// TIA Portal V17 export
// export: Created 2026-04-13T11:12:41.3915704Z, ExportSetting WithDefaults, DisplayName Totally Integrated Automation Portal, DisplayVersion V17 Update 4, DisplayName TIA Portal Openness, DisplayVersion V17 Update 4, DisplayName TIA Portal Version Control Interface, DisplayVersion V17, DisplayName SINAMICS Startdrive Advanced, DisplayVersion V17, DisplayName SINAMICS Startdrive G130, G150, S120, S150, SINAMICS MV, S210, DisplayVersion V17, DisplayName SINAMICS Startdrive G110M, G120, G120C, G120D, G120P, G115D, DisplayVersion V17, DisplayName STEP 7 Professional, DisplayVersion V17 Update 4, DisplayName STEP 7 Safety, DisplayVersion V17, DisplayName WinCC Professional, DisplayVersion V17 Update 4
FUNCTION_BLOCK "A1-台达DTC"   // FB33, SCL
{ S7_Optimized_Access := 'TRUE' }
VERSION : 0.1
// stored: AutoNumber true, IsIECCheckEnabled false, IsRetainMemResEnabled false, MemoryReserve 100, SetENOAutomatically false, UDAEnableTagReadback false
   VAR_INPUT
      站号 : UInt;
      触发 : Bool;
      输入模式 : Int;
      输入开关 : Bool;
      A输入设定 : Real;
      输入开度 : Real;
   END_VAR
   VAR_OUTPUT
      结束 : Bool;
      高高报警 : Bool;
      高报警 : Bool;
      低报警 : Bool;
      低低报警 : Bool;
      传感器故障 : Bool;
      输出控制P : Real;
      输出控制I : Real;
      输出控制D : Real;
      输出开度读 : Real;
   END_VAR
   VAR_IN_OUT
      B当前量 : Real;
      输入设定读 : Real;
      输出模式读 : Real;
      高高报设置 : Real;
      高报设置 : Real;
      低报设置 : Real;
      低低报设置 : Real;
      自整定开关 : Bool;
      Modbus_Master_Instance : Modbus_Master;
   END_VAR
   VAR DB_SPECIFIC
      当前指令ID : Int;
      上一次指令ID : Int;
      modbus_data : Struct
         触发 : Bool;
         站号 : UInt;
         模式 : USInt;
         地址 : UDInt;
         数据长度 : UInt;
         完成 : Bool;
         忙碌 : Bool;
         出错 : Bool;
         故障码 : Word;
         数据缓存区 : Array[1..50] of Word;
      END_STRUCT;
      报错代码 : Array[1..20] of Word;
      进温P读 : Int;
      进温I读 : Int;
      进温D读 : Int;
      T1_SV_写 : Int;
      进温AT开关 : Bool;
      进温AT开关_bak : Bool;
      进温AT_写字 : UInt;
      进温AT_读字 : UInt;
      T1_P值比对1 : Int;
      T1_P值比对2 : Int;
      进温启停字 : UInt;
      T1 { S7_SetPoint := 'True'} : TON_TIME;
   END_VAR
   VAR_TEMP
      tm_int : Int;
      tm_real : Real;
   END_VAR
BEGIN
   //程序1

   IF #触发 THEN
       #当前指令ID := 1;
   END_IF;

   #modbus_data.站号 := #站号;

   IF #当前指令ID = 9 THEN
       IF #进温AT_写字 = #进温AT_读字 THEN
           #当前指令ID := 10;
       END_IF;
   END_IF;

   CASE #当前指令ID OF
       1:
           //读取地址44097-44098
           #modbus_data.模式 := 0;
           #modbus_data.地址 := 44097;
           #modbus_data.数据长度 := 2;
       2:
           //读取地址44102
           (* 1005H-4101-44102  默认0   控制方式 0：PID；1：ON/OFF；2：手动；3：PID 过程控制 *)
           #modbus_data.模式 := 0;
           #modbus_data.地址 := 44102;
           #modbus_data.数据长度 := 1;
       3:
           //读取地址44106-44108
           (*  
           1009H-4105-44106  默认476 PB 比例带设定值 1 ~ 9,999, 温度单位为 0.1 度，模拟输入为 1EU
           100AH-4106-44107  默认260 Ti 积分控制常量设定值 0 ~ 9,999
           100BH-4107-44108  默认41 Td 微分控制常量设定值 0 ~ 9,999 *)
           #modbus_data.模式 := 0;
           #modbus_data.地址 := 44106;
           #modbus_data.数据长度 := 3;
       4:
           //读取地址44116
           (* 1013H-4115-44116  默认0   输出 2 输出量读取与写入 单位为 0.1%，写入只在手动控制模式下有效（DTC1000/2000 机种） *)
           #modbus_data.模式 := 0;
           #modbus_data.地址 := 44116;
           #modbus_data.数据长度 := 1;
       5:
           //读取地址12068
           (* 0813H-2067-12068  读写自动调谐状态 自动调谐停止：0（预设），自动调谐开始：1 *)
           #modbus_data.模式 := 0;
           #modbus_data.地址 := 12068;
           #modbus_data.数据长度 := 1;
       6:
           //写入地址44098
           (* 1001H-4097-44098       默认0 "SV" 设定值 温度以 0.1 度为计量单位，模拟输入为 1EU。 *)
           #tm_real := #A输入设定 * 10.0;
           #T1_SV_写 := REAL_TO_INT(#tm_real);
           #modbus_data.数据缓存区[1] := INT_TO_WORD(#T1_SV_写);
           #modbus_data.模式 := 1;
           #modbus_data.地址 := 44098;
           #modbus_data.数据长度 := 1;
       7:
           //写入地址44102
           (* 1005H-4101-44102  默认0   控制方式 0：PID；1：ON/OFF；2：手动；3：PID 过程控制 *)
           #modbus_data.数据缓存区[1] := INT_TO_WORD(#输入模式);
           #modbus_data.模式 := 1;
           #modbus_data.地址 := 44102;
           #modbus_data.数据长度 := 1;
       8:
           //写入地址44116
           (* 1013H-4115-44116  默认0   输出 2 输出量读取与写入 单位为 0.1%，写入只在手动控制模式下有效（DTC1000/2000 机种） *)
           #tm_real := #输入开度 * 10;
           #tm_int := REAL_TO_INT(#tm_real);
           #modbus_data.数据缓存区[1] := INT_TO_WORD(#tm_int);
           #modbus_data.模式 := 1;
           #modbus_data.地址 := 44116;
           #modbus_data.数据长度 := 1;
       9:
           //写入地址2068
           (* 0813H-2067-12068  读写自动调谐状态 自动调谐停止：0（预设），自动调谐开始：1 *)

           #modbus_data.数据缓存区[1] := UINT_TO_WORD(#进温AT_写字);
           #modbus_data.模式 := 1;
           #modbus_data.地址 := 2068;
           #modbus_data.数据长度 := 1;
       10:
           //写入地址2069
           (* 0814H-2068-12069  控制执行/停止设定 0：停止，1：执行（预设） *)
           #modbus_data.数据缓存区[1] := UINT_TO_WORD(#进温启停字);
           #modbus_data.模式 := 1;
           #modbus_data.地址 := 2069;
           #modbus_data.数据长度 := 1;

   END_CASE;




   #modbus_data.触发 := #当前指令ID <> #上一次指令ID;
   #上一次指令ID := #当前指令ID;



   //程序2


   #Modbus_Master_Instance(REQ := #modbus_data.触发,
                           MB_ADDR := #modbus_data.站号,
                           MODE := #modbus_data.模式,
                           DATA_ADDR := #modbus_data.地址,
                           DATA_LEN := #modbus_data.数据长度,
                           DONE => #modbus_data.完成,
                           BUSY => #modbus_data.忙碌,
                           ERROR => #modbus_data.出错,
                           STATUS => #modbus_data.故障码,
                           DATA_PTR := #modbus_data.数据缓存区);

   //程序3

   IF #modbus_data.完成 THEN
       CASE #当前指令ID OF
           1:
               //44097
               (* 1000H-4096-44097       PV 目前测量值
               （温度以 0.1 刻度为计量单位，模拟输入为 1EU。
               下列读值表示错误发生：
               8002H（32770） 输入读值尚未取得
               8003H（32771） 未接传感器
               8004H（32772） 传感器型式错误
               8006H（34774） 输入值无法测量,输入 ADC 错误
               8007H（32775） 内存无法读写） *)
               #tm_int := WORD_TO_INT(#modbus_data.数据缓存区[1]);
               #tm_real := INT_TO_REAL(#tm_int);
               #B当前量 := #tm_real / 10;
               //44098
               #tm_int := WORD_TO_INT(#modbus_data.数据缓存区[2]);
               #tm_real := INT_TO_REAL(#tm_int);
               #输入设定读 := #tm_real / 10;

           2:
               //44102
               (* 1005H-4101-44102  默认0   控制方式 0：PID；1：ON/OFF；2：手动；3：PID 过程控制 *)
               #tm_int := WORD_TO_INT(#modbus_data.数据缓存区[1]);
               #输出模式读 := #tm_int;
           3:
               (*   1009H-4105-44106  默认476 PB 比例带设定值 1 ~ 9,999, 温度单位为 0.1 度，模拟输入为 1EU
                    100AH-4106-44107  默认260 Ti 积分控制常量设定值 0 ~ 9,999
                    100BH-4107-44108  默认41 Td 微分控制常量设定值 0 ~ 9,999 *)
                    //44106
                    #tm_int := WORD_TO_INT(#modbus_data.数据缓存区[1]);
                    #进温P读 := #tm_int;
                    //44107
                    #tm_int := WORD_TO_INT(#modbus_data.数据缓存区[2]);
                    #进温I读 := #tm_int;
                    //44108
                    #tm_int := WORD_TO_INT(#modbus_data.数据缓存区[3]);
                    #进温D读 := #tm_int;
                4:
                    //44116
                    (* 1013H-4115-44116  默认0   输出 2 输出量读取与写入 单位为 0.1%，写入只在手动控制模式下有效（DTC1000/2000 机种） *)
                    #tm_int := WORD_TO_INT(#modbus_data.数据缓存区[1]);
                    #tm_real := INT_TO_REAL(#tm_int);
                    #输出开度读 := #tm_real / 10;
                5:
                    //12068
                    (* 0813H-2067-12068  读写自动调谐状态 自动调谐停止：0（预设），自动调谐开始：1 *)
                    #进温AT_读字 := WORD_TO_UINT(#modbus_data.数据缓存区[1]);
            END_CASE;
        END_IF;

        IF #modbus_data.出错 AND #当前指令ID > 0 AND #当前指令ID < 12 THEN
            #报错代码[#当前指令ID] := #modbus_data.故障码;
        END_IF;

        IF #modbus_data.完成 OR #modbus_data.出错 THEN
            #当前指令ID := #当前指令ID + 1;
        END_IF;

        IF #当前指令ID > 10 THEN
            #当前指令ID := 0;
            #上一次指令ID := 0;
            #结束 := 1;
        ELSE
            #结束 := 0;
        END_IF;

        //程序4

        IF NOT #自整定开关 THEN
            #进温AT_写字 := 0;
            #T1_P值比对1 := #进温P读;
            #T1_P值比对2 := #进温P读;
        END_IF;
        IF #自整定开关 THEN

            #进温AT_写字 := 65280;

            #T1_P值比对2 := #进温P读;
        END_IF;
        IF #T1_P值比对1 <> #T1_P值比对2 THEN
            #自整定开关 := 0;
        END_IF;

        //程序5


        IF #自整定开关 THEN
            #进温AT_写字 := 16#FF00;
        ELSE
            #进温AT_写字 := 16#0;
        END_IF;

        IF #输入开关 THEN
            #进温启停字 := 16#FF00;
        ELSE
            #进温启停字 := 16#0;
        END_IF;

       //程序6

        #输出控制P := INT_TO_REAL(#进温P读);
        #输出控制I := INT_TO_REAL(#进温I读);
        #输出控制D := INT_TO_REAL(#进温D读);

        //报警
        IF #B当前量 > #高报设置 THEN
            #高报警 := 1;
        ELSE
            #高报警 := 0;
        END_IF;

        IF #B当前量  > #高高报设置 THEN
            #高高报警 := 1;
        ELSE
            #高高报警 := 0;
        END_IF;

        IF #B当前量 < #低报设置 THEN
            #低报警 := 1;
        ELSE
            #低报警 := 0;
        END_IF;

        IF #B当前量 < #低低报设置 THEN
            #低低报警 := 1;
        ELSE
            #低低报警 := 0;
        END_IF;

        IF #B当前量 > 500 AND #B当前量 < -10 THEN
            #传感器故障 := 1;
        ELSE
            #传感器故障 := 0;
        END_IF;
END_FUNCTION_BLOCK
